// TIA Portal V20 export
DATA_BLOCK "IDB_ToteTracking"   // DB11
// stored: InstanceOfName ProductionLine.FB_ToteTracking, InstanceOfType FB, Namespace ProductionLine
"ProductionLine.FB_ToteTracking"
   // VAR
   //    ZoneBpJam_Occ : TON_TIME;
   //    ZoneBpJam_NotOcc { S7_SetPoint := 'True'} : TON_TIME;
   //    DivertToManual { S7_SetPoint := 'True'} : Bool;
   //    HoldDivertToManual : Bool;
   //    RT_Exit_1_ : Array[1..1] of R_TRIG;
   //    RT_Exit_2_ : Array[1..6] of R_TRIG;
   //    NoReadTote { S7_SetPoint := 'True'} : String;
   //    NoData : Array[1..6] of Bool;
   // END_VAR
BEGIN
END_DATA_BLOCK
